(* PLC project BlogProject.project, CODESYS CODESYS V3.5 SP14 Patch 3 *)
(* stored: creationDateTime 2021-10-07T21:06:18.7753655, modificationDateTime 2021-10-07T20:40:20.1109198 *)

FUNCTION_BLOCK mcIsSystemStopCommand IMPLEMENTS itfEvent
  VAR
    bStopCommand : BOOL;
  END_VAR

            
          

METHOD getEvent : BOOL
                  getEvent:=StopCommand;
                
END_METHOD
END_FUNCTION_BLOCK
